FUNCTION_BLOCK controller
  (* Standard: 61499-2 *)
  (* Version 0.1, 2017-00-25, hpea485, UOA *)
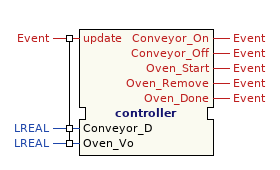
  EVENT_INPUT
    update WITH Conveyor_D, Oven_Vo;
  END_EVENT
  EVENT_OUTPUT
    Conveyor_On;
    Conveyor_Off;
    Oven_Start;
    Oven_Remove;
    Oven_Done;
  END_EVENT
  VAR_INPUT
    Conveyor_D : LREAL;
    Oven_Vo : LREAL;
  END_VAR
  VAR
    Dstart : LREAL;
  END_VAR
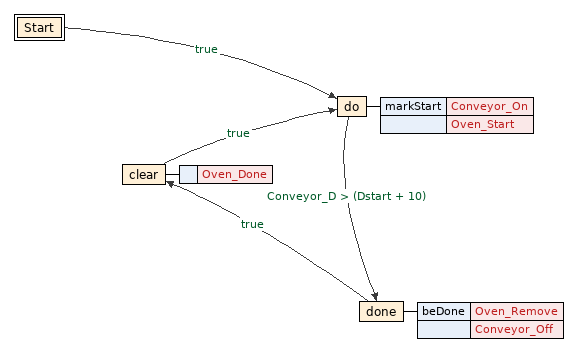
  EC_STATES
    Start;
    do : markStart -> Conveyor_On, -> Oven_Start;
    done : beDone -> Oven_Remove, -> Conveyor_Off;
    clear : -> Oven_Done;
  END_STATES
  EC_TRANSITIONS
    Start TO do := true;
    do TO done := Conveyor_D > (Dstart + 10);
    done TO clear := true;
    clear TO do := true;
  END_TRANSITIONS
  ALGORITHM markStart IN C:
me->Dstart = me->Conveyor_D;
  END_ALGORITHM
  ALGORITHM beDone IN C:
//printf("Pizza cooked, temperature is %f yum yum\n", me->Oven_Vo);
  END_ALGORITHM
END_FUNCTION_BLOCK
